(*udt (user defined type) of Beckhoff EP9214 IP67 Block - Power Distribution Block, individual channel data:
	To work in conjunction of udt_EP9214_STAT_yyyymmdd
	auth. Brent Lekx-Toniolo, copy/paste from 9224 from r.jones of Sodecia GTAC; 

------------------------------------------------------------------------
REVISION NOTES:
	Version 20250704
		- Initial Concept
------------------------------------------------------------------------

*)


TYPE udt_EP9214_DEV_CMD_20250704 :
STRUCT

	Enable_Control_Via_Fieldbus: BOOL;
	Global_Reset: BOOL;

END_STRUCT
END_TYPE

(* stored: Version 1.1.0.1, ProductVersion 3.1.4024.12
   DUT udt_EP9214_DEV_CMD_20250704: Id {52a0dd59-4568-411b-bb07-c3aa5422f318} *)
